FUNCTION_BLOCK FB_Drilling
VAR_INPUT
	ins_CommIn				:Type_CommIn_Drilling;
	inm_Reset				:BOOL;
	inint_Position			:INT;
END_VAR
VAR_OUTPUT
	outs_CommOut				:Type_CommOut_Drilling;
	o_AverageCycleTime			:REAL;
END_VAR
VAR
	o_TotalCycleTime		:BYTE;
	
	o_PartExists			 :BOOL;
	o_Drilling_Done 		 :BOOL;
	o_ProcessCycleTime			:REAL;
	
	m_BaseFinished 	:BOOL;
	m_First			:BOOL;
	m_FirstCycleTime			:BOOL;
	
	RetVal 			: enum_RetVal;
	
	
	(* Timers *)
	SFCInit			:BOOL;
	
	T03_Locate_Drill_Spots 		:TON;
	T04_Drilling_Process 		:TON;
	T05_Filling_Off 			:TON;
	
	Instance_CountTotalCycleTime		:FB_CountCycleTime();
	Instance_CountProcessCycleTime		:FB_CountCycleTime();
	
	
END_VAR


IF inm_Reset = FALSE
	THEN
	SFCReset:=FALSE;
	A01_AutomaticMode();
	
	ELSE
		SFCReset:=TRUE;
		A01_AutomaticMode();
END_IF

ACTION A01_AutomaticMode:
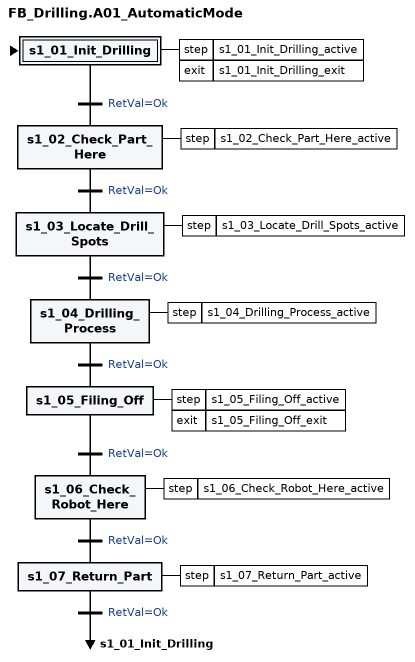
INITIAL_STEP s1_01_Init_Drilling:
    s1_01_Init_Drilling_active(N);  // step action
    s1_01_Init_Drilling_exit(P0);  // exit action
END_STEP
TRANSITION FROM s1_01_Init_Drilling TO s1_02_Check_Part_Here
    := RetVal=Ok;
END_TRANSITION
STEP s1_02_Check_Part_Here:
    s1_02_Check_Part_Here_active(N);  // step action
END_STEP
TRANSITION FROM s1_02_Check_Part_Here TO s1_03_Locate_Drill_Spots
    := RetVal=Ok;
END_TRANSITION
STEP s1_03_Locate_Drill_Spots:
    s1_03_Locate_Drill_Spots_active(N);  // step action
END_STEP
TRANSITION FROM s1_03_Locate_Drill_Spots TO s1_04_Drilling_Process
    := RetVal=Ok;
END_TRANSITION
STEP s1_04_Drilling_Process:
    s1_04_Drilling_Process_active(N);  // step action
END_STEP
TRANSITION FROM s1_04_Drilling_Process TO s1_05_Filing_Off
    := RetVal=Ok;
END_TRANSITION
STEP s1_05_Filing_Off:
    s1_05_Filing_Off_active(N);  // step action
    s1_05_Filing_Off_exit(P0);  // exit action
END_STEP
TRANSITION FROM s1_05_Filing_Off TO s1_06_Check_Robot_Here
    := RetVal=Ok;
END_TRANSITION
STEP s1_06_Check_Robot_Here:
    s1_06_Check_Robot_Here_active(N);  // step action
END_STEP
TRANSITION FROM s1_06_Check_Robot_Here TO s1_07_Return_Part
    := RetVal=Ok;
END_TRANSITION
STEP s1_07_Return_Part:
    s1_07_Return_Part_active(N);  // step action
END_STEP
TRANSITION FROM s1_07_Return_Part TO s1_01_Init_Drilling
    := RetVal=Ok;
END_TRANSITION
END_ACTION

ACTION s1_01_Init_Drilling_active:
RetVal:=Running;
Instance_CountTotalCycleTime(inm_TimeActive:=FALSE);
o_TotalCycleTime:=REAL_TO_BYTE(Instance_CountTotalCycleTime.outr_CycleTime);

outs_CommOut.s_Robot.m_Empty:=TRUE;
outs_CommOut.s_Robot.m_Ready:=FALSE;

IF  ins_CommIn.s_Robot.m_OutOfArea
	THEN
	Instance_CountTotalCycleTime(inm_TimeActive:=TRUE);	
	RetVal:=Ok;
END_IF
END_ACTION

ACTION s1_01_Init_Drilling_exit:
IF NOT m_FirstCycleTime
	THEN
	o_AverageCycleTime := 30;
END_IF
END_ACTION

ACTION s1_02_Check_Part_Here_active:
RetVal:=Running;

IF ins_CommIn.s_Robot.m_OutOfArea = FALSE(*Daca position[2] e true inseamna ca robotul e in pozitie, dar nu s-a facut place!!	*)
	AND ins_CommIn.s_Robot.m_Work = FALSE	
	THEN
	outs_CommOut.s_Robot.m_Empty:=FALSE;	
END_IF

IF ins_CommIn.s_Robot.m_PartDropped
	THEN
	Instance_CountProcessCycleTime(inm_TimeActive:=TRUE);
	RetVal:=Ok;
END_IF
END_ACTION

ACTION s1_03_Locate_Drill_Spots_active:
RetVal:=Running;

T03_Locate_Drill_Spots(IN:=TRUE,PT:=T#1S,Q=>,ET=>);

IF T03_Locate_Drill_Spots.Q
	THEN
	T03_Locate_Drill_Spots(IN:=FALSE);
	RetVal:=Ok;
END_IF
END_ACTION

ACTION s1_04_Drilling_Process_active:
RetVal:=Running;

T04_Drilling_Process(IN:=TRUE,PT:=T#28S,Q=>,ET=>);

IF T04_Drilling_Process.Q
	THEN
	T04_Drilling_Process(IN:=FALSE);
	RetVal:=Ok;
END_IF
END_ACTION

ACTION s1_05_Filing_Off_active:
RetVal:=Running;

T05_Filling_Off(IN:=TRUE,PT:=T#1S,Q=>,ET=>);

IF T05_Filling_Off.Q
	THEN
	Instance_CountProcessCycleTime(inm_TimeActive:=FALSE);
	o_ProcessCycleTime:=Instance_CountProcessCycleTime.outr_CycleTime;
	
	IF m_First 
	THEN
		o_AverageCycleTime := (o_AverageCycleTime + o_ProcessCycleTime)/2;
		ELSE
		o_AverageCycleTime := o_ProcessCycleTime;
	END_IF
	o_PartExists:=TRUE;
	outs_CommOut.s_Robot.m_Ready:=TRUE;
	T05_Filling_Off(IN:=FALSE);
	RetVal:=Ok;
END_IF
END_ACTION

ACTION s1_05_Filing_Off_exit:
m_First:=TRUE;
END_ACTION

ACTION s1_06_Check_Robot_Here_active:
RetVal:=Running;

IF ins_CommIn.s_Robot.m_OutOfArea=FALSE
	THEN 
	RetVal:=Ok;	
END_IF
END_ACTION

ACTION s1_07_Return_Part_active:
RetVal:=Running;
m_FirstCycleTime:=TRUE;
o_PartExists:=FALSE;

IF ins_CommIn.s_Robot.m_Work=FALSE
	AND ins_CommIn.s_Robot.m_PartDropped=FALSE
	THEN
	RetVal:=Ok;
END_IF


(*	Aici piesa este finalizata si ea trebuie transportata la urmatorul modul

		=> 		Pick aici ---> Place Pe Metalization 
		*)
END_ACTION

ACTION s2_01_Base_Move_active:
IF NOT m_BaseFinished
THEN
	RetVal := OK;
ELSE
	RetVal := RUNNING;
END_IF
END_ACTION

END_FUNCTION_BLOCK

(* stored: Version 1.1.0.1, ProductVersion 3.1.4024.3
   POU FB_Drilling: Id {cecdbc68-d18e-4716-bd51-1af734f02f1b}, SpecialFunc None
   Folder S1: Id {e6995024-f40a-4c3a-988f-4b61d2466107}
   Folder S2: Id {d0b11b46-f2bf-4e8f-a363-a45bcf70e2df}
   Action A01_AutomaticMode: Id {6bc7e114-c67e-44a8-af29-ee3db5e59db8}
   Action s1_01_Init_Drilling_active: Id {3b821f26-1a9e-456c-96dd-efd7fa358d7a}
   Action s1_01_Init_Drilling_exit: Id {f37cd5b0-7c0b-4b9c-a062-c2422f371e58}
   Action s1_02_Check_Part_Here_active: Id {342e7b19-2a57-45c2-840d-508c0bbbbbfb}
   Action s1_03_Locate_Drill_Spots_active: Id {15279863-0aea-4a39-b542-6c3b96a09535}
   Action s1_04_Drilling_Process_active: Id {1c14c5bb-83be-4a6f-b264-374e4856e17a}
   Action s1_05_Filing_Off_active: Id {e5564286-d7f4-431c-ac26-4d4541394894}
   Action s1_05_Filing_Off_exit: Id {011bb6de-b150-4965-94a9-7e18c370b52e}
   Action s1_06_Check_Robot_Here_active: Id {440103ce-5a35-4166-852a-8cd3ca32b4f3}
   Action s1_07_Return_Part_active: Id {c63b6a75-37cd-4bb9-aad9-a8beae046671}
   Action s2_01_Base_Move_active: Id {b8fb6fd6-e4c4-4d89-adb6-214715539927} *)
